{attribute 'qualified_only'}
VAR_GLOBAL CONSTANT
	HEADER_STRING_SIZE : UDINT := 1024; 
	PAYLOAD_STRING_SIZE : UDINT := 8000; // typically 1/8th of the Runtime Stack Size
END_VAR

(* stored: Version 1.1.0.1, ProductVersion 3.1.4024.12
   GVL ServerConfiguration: Id {9a1f076d-eeae-4f72-ae58-e87939461d63}, ParameterList True *)
